FUNCTION F_WRITE_LOG : BOOL
VAR_INPUT
	inputColor: ST_LED; 
	status: STRING;
END_VAR
VAR
	stLOG: ST_Log := (sStatus:=CONCAT(CONCAT(status, ' -'), inputColor.color)); //log to be added to the log collection
END_VAR

stLog.sTime := EMPTY.tTime;
F_WRITE_MEMORY(cbData:=SIZEOF(stLog),pData:=ADR(stLog),cbBuffer:=SIZEOF(MAIN.stSystem.arrLog),pBuffer:=ADR(MAIN.stSystem.arrLog));

END_FUNCTION

(* stored: Version 1.1.0.1, ProductVersion 3.1.4022.12
   POU F_WRITE_LOG: Id {b70c0d0e-64b6-48e2-a10d-88c7e228e0d9}, SpecialFunc None *)
